{attribute addProperty BoxType "EL7031-0030-0016"}
{attribute addProperty Id "UnderrangeAT %I*BOOL811OverrangeAT %I*BOOL812Limit_xAT %I*ARRAY[0 ..1] OF BYTE1620TxPDO_ToggleAT %I*BOOL8116ValueAT %I*INT16217"}
{attribute addProperty CRC "2250630994"}
{attribute addProperty SizeInBites "56"}
{attribute addProperty SizeInBytes "7"}
TYPE AI_Standard_Channel_5B3BB325 :
STRUCT
	{attribute addProperty Name "Underrange"}
	Underrange AT %I* : BOOL;
	{attribute addProperty Name "Overrange"}
	Overrange AT %I* : BOOL;
	{attribute addProperty Name "Limit"}
	Limit_x AT %I* : ARRAY[0 ..1] OF BYTE;
	{attribute addProperty Name "TxPDO_Toggle"}
	TxPDO_Toggle AT %I* : BOOL;
	{attribute addProperty Name "Value"}
	Value AT %I* : INT;
END_STRUCT
END_TYPE

(* stored: Version 1.2.0.0, ProductVersion 3.1.4024.9
   DUT AI_Standard_Channel_5B3BB325: Id {7da6dfd1-fb73-4c30-9194-688356a367d0} *)
